PROGRAM Initialize
VAR
END_VAR

// go to the initial position (0,0,0,0)
IF NOT IO.Initialized THEN
	IF IO.EndRotationSensor THEN
		IO.MotorRotation := 0;
		IO.MotorRotationDirection := 0;
		Automatic.RCurrentlyMoving := FALSE;
	ELSE 
		IO.MotorRotationDirection := 1;
		Automatic.RCurrentlyMoving := TRUE;
		IO.MotorRotation := 1;
	END_IF
	
	IF IO.EndLiftingSensor THEN
		IO.MotorLifting := 0;
		IO.MotorLiftingDirection := 0;
		Automatic.LCurrentlyMoving := FALSE;
	ELSE 
		IO.MotorLiftingDirection := 1;
		Automatic.LCurrentlyMoving := TRUE;
		IO.MotorLifting := 1;
	END_IF
	
	IF IO.EndExtensionSensor THEN
		IO.MotorExtension := 0;
		IO.MotorExtensionDirection := 0;
		Automatic.ECurrentlyMoving := FALSE;
	ELSE 
		IO.MotorExtensionDirection := 1;
		Automatic.ECurrentlyMoving := TRUE;
		IO.MotorExtension := 1;
	END_IF
	
	IF IO.EndGripSensor THEN
		IO.MotorGrip := 0;
		IO.MotorGripDirection := 0;
		Automatic.GCurrentlyMoving := FALSE;
	ELSE 
		IO.MotorGripDirection := 1;
		Automatic.GCurrentlyMoving := TRUE;
		IO.MotorGrip := 1;
	END_IF
		
	IF IO.EndRotationSensor AND IO.EndLiftingSensor AND IO.EndExtensionSensor AND IO.EndGripSensor THEN
		Automatic.RCurrentlyMoving := FALSE;
		Automatic.ECurrentlyMoving := FALSE;
		Automatic.LCurrentlyMoving := FALSE;
		Automatic.GCurrentlyMoving := FALSE;
		IO.Initialized := TRUE;
		IO.PreviousManualMode := TRUE;
	END_IF
END_IF

END_PROGRAM

(* stored: Version 1.1.0.1, ProductVersion 3.1.4024.13
   POU Initialize: Id {acc585e9-1428-4ae4-802a-0f449af0d289}, SpecialFunc None *)
